SUBAPPLICATION R_AR_SUB (* Subtrahiert einen AR-Wert von einem festen REAL-Minuenden (OUT = MINUEND - IN; kein zweiter AR-Socket noetig - der Minuend wird per Parameter bei der Instanziierung eingebacken) *)
  (* Standard: 61499-2 *)
  (* Version 1.0, 2026-09-27, Franz Höpfinger, Meisterschulen am Ostbahnhof *)
  PACKAGE MyLib::sys;
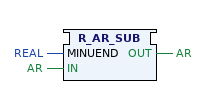
  VAR_INPUT
    MINUEND : REAL := REAL#0.0; (* Fester Minuend, ueber Parameter bei der Instanziierung gesetzt *)
  END_VAR
  SOCKETS
    IN : adapter::types::unidirectional::AR; (* Zu subtrahierender Subtrahend *)
  END_SOCKETS
  PLUGS
    OUT : adapter::types::unidirectional::AR; (* MINUEND - IN *)
  END_PLUGS
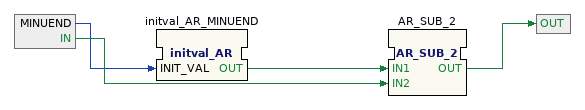
  FBS
    initval_AR_MINUEND : adapter::types::unidirectional::AR::initval::initval_AR;
    AR_SUB_2 : adapter::iec61131::arithmetic::AR_SUB_2;
  END_FBS
  DATA_CONNECTIONS
    MINUEND TO initval_AR_MINUEND.INIT_VAL;
  END_CONNECTIONS
  ADAPTER_CONNECTIONS
    initval_AR_MINUEND.OUT TO AR_SUB_2.IN1;
    IN TO AR_SUB_2.IN2;
    AR_SUB_2.OUT TO OUT;
  END_CONNECTIONS
END_SUBAPPLICATION
